Staubli VAL3: iocWriteBack.pgx

program iocWriteBack(string XsResponse (dimensions=1))
begin
  //
  //header begin
  // PROGRAM iocWriteBack()
  //
  // pgm writes text via TCP/IP to IOC client socket on CS8
  //
  // input parms:
  //    XsResponse = string passed from calling program
  //
  // output parms:
  //    none
  //
  // called from:  iocCmdHandler()
  //
  // initial release:  KN
  // Release 2:  KN
  //  changed functionality from CS8 host to CS8 client
  //  updated documentation
  //header end
  //
  sioIOCclient=XsResponse
end
